//==================================================================================================
//							Beckhoff Automation Poland
//									14.03.2023
//
// Code owner: TG
//
// Function block for processing digital outputs. 
// Includes filters, simulating, various operational modes selection and edges detection.
//
// Used libraries: 
//	Tc2_standard						|| 3.3.3.0
//
// Used FBs:
//
// Used DUTs:
//
//  v1.0	|| TC v 3.1.4024.40		|| First edition
//==================================================================================================
FUNCTION_BLOCK FB_DigitalOutput
VAR
	Out 					AT %Q* 				: BOOL;
	bManualIn									: BOOL;		// HMI
	
	{attribute 'hide'}
	bManualMode_Internal						: BOOL;		// Internal flag - active when manual mode selected
	_bIn										: BOOL;
	{attribute 'hide'}
	_bOut										: BOOL; 
	{attribute 'hide'}
	_tTimeDelay									: TIME;
	{attribute 'hide'}
	_tTimeOn									: TIME;
	{attribute 'hide'}
	_tTimeOff									: TIME;
	{attribute 'hide'}
	_nMode										: DINT;															
END_VAR

CASE nMode OF							//case regarding mode selection 

	0:	// false
		Off();
	
	1:	// true
		On();

	2:	// auto normal
		Auto();
		
	9:	// manual
		Manual();
	
	10:	// clock
		Clock();

	11: // min OFF, min ON	
		MinOnOff();	
	
	20: // single TP
		SingleTP();
	
	21: // single TON
		SingleTON();	
							
	30: // mutli TP
		MultiTP();

	31:	// mutli TON
		MultiTON();
		
ELSE		
	Off();
	
		
END_CASE;

METHOD Auto 									: BOOL							//output actual value 
VAR_INPUT
END_VAR
bOut											:= bIn;

bManualMode_Internal							:= FALSE;
END_METHOD

PROPERTY bIn 									: BOOL								//value before processing
GET
bIn												:=_bIn;
END_GET
SET
_bIn											:= bIn;
END_SET
END_PROPERTY

PROPERTY bOut 									: BOOL							//processed output value
GET
bOut											:= _bOut;
END_GET
SET
_bOut											:= bOut;
Out												:= bOut;
END_SET
END_PROPERTY

METHOD Clock 									: BOOL							//use output for specifed time with pause between
VAR_INST
	{attribute 'hide'}
	tonTimer									: TON;
END_VAR
tonTimer(IN := NOT tonTimer.Q,
		PT										:= tTimeOn + tTimeOff);
bOut											:= tonTimer.ET <  tTimeOn;
		
bManualMode_Internal							:= FALSE;
END_METHOD

METHOD Manual 									: BOOL							//Control output value manually
IF bManualMode_Internal THEN
	bOut										:= bManualIn;
ELSE
	bManualIn									:= bOut;
END_IF

bManualMode_Internal							:= TRUE;
END_METHOD

METHOD ManualEx 								: BOOL							//Control output value manually
VAR_INPUT
	bIn											: BOOL;
END_VAR
bOut											:= bIn;

bManualMode_Internal							:= FALSE;
END_METHOD

METHOD MinOnOff 								: BOOL						//output with specific active and disabled time
VAR_INST
	TimeMinOn									: TON;
	TimeMinOff									: TON;	
END_VAR
TimeMinOff(IN := NOT bOut, PT := tTimeOff);			
                        						
TimeMinOn(IN := bOut, PT := tTimeOn);	
		
IF TimeMinOn.Q THEN
	bOut										:= bIn;
END_IF;			
		
IF TimeMinOff.Q THEN
	bOut										:= bIn;
END_IF;

bManualMode_Internal							:= FALSE;
END_METHOD

METHOD MultiTON 								: BOOL						//activation delay dependent from value
VAR_INST
	Timer										: TON;
END_VAR
Timer(IN := bIn, PT := tTimeDelay);

bOut											:= Timer.Q;

bManualMode_Internal							:= FALSE;
END_METHOD

METHOD MultiTP 									: BOOL							//pulse dependent from value
VAR_INST
	Timer										: TP;
END_VAR
Timer(IN := bIn, PT := tTimeOn);
		
bOut											:= Timer.Q;

bManualMode_Internal							:= FALSE;
END_METHOD

PROPERTY nMode 									: DINT							//mode selection value: 0- false 1-true 2 - auto_normal, 10- clock, 20 - single tp, 21 - single ton, 9 - manual, 30 - multi tp, 31 - multi ton, 11 - min ON, min OFF
GET
nMode											:= _nMode;
END_GET
SET
_nMode											:= nMode;
END_SET
END_PROPERTY

METHOD Off 										: BOOL								//set value FALSE
bOut											:= FALSE;

bManualMode_Internal							:= FALSE;
END_METHOD

METHOD On 										: BOOL								//set value TRUE
bOut											:= TRUE;

bManualMode_Internal							:= FALSE;
END_METHOD

METHOD SingleTON 								: BOOL						//activation delay 
VAR_INST
	Timer										: TON;
END_VAR
Timer(IN := TRUE, PT := tTimeDelay);

bOut											:= Timer.Q;

bManualMode_Internal							:= FALSE;
END_METHOD

METHOD SingleTP 								: BOOL						//single pulse
VAR_INST
	Timer										: TP;
END_VAR
Timer(IN := TRUE, PT := tTimeOn);

bOut											:= Timer.Q;

bManualMode_Internal							:= FALSE;
END_METHOD

PROPERTY tTimeDelay  								: TIME						//delay time in [ms], for Single/MultiTON mode
GET
tTimeDelay										:= _tTimeDelay;
END_GET
SET
_tTimeDelay										:= tTimeDelay;
END_SET
END_PROPERTY

PROPERTY tTimeOff 								: TIME						//minimum output on time [ms], for minOnOff mode
GET
tTimeOff										:= _tTimeOff;
END_GET
SET
_tTimeOff										:= tTimeOff;
END_SET
END_PROPERTY

PROPERTY tTimeOn 								: TIME						//minimum output off time [ms], for minOnOff mode
GET
tTimeOn											:=_tTimeOn;
END_GET
SET
_tTimeOn										:= tTimeOn;
END_SET
END_PROPERTY

END_FUNCTION_BLOCK

(* stored: Version 1.1.0.1, FileIdentifier 9c9296da76f6555697687ec98103123ce9290b24, FileSignature 4b7ff2dcf8c12612268e668eaf2997718c55023cd67da2f5992bdf710eefc9968962d0b293f44ff252512e4510ae557b74a6a527a16271f1788755e7e6d9445defe0fe348b14a65da049c3d86c0c9e8fdd809d3d46764a5bcdca4ca8c0c737abe1dca42b05d38a2eedf13d4ff265bcc4314e1f238197d24dcd4ab5bd84eb4ef6208a6f210ed1960d85d639d221da18380a7ed45771d073b4f8f16abf18f4a0101355f8787fddc439370796d36f83c19f69321c38f61acdb8ad15c808a511caa439041c93119310479aa3316171e14b610b326d88d603c3c53c91d3b49ea8358598d3b6d06331ac0704becd62f57d1ee26a41c64ff01206e21afefac73dbd0c3d
   POU FB_DigitalOutput: Id {b9e9f56b-5870-4da1-94e5-b2a4388e6247}, SpecialFunc None
   Folder Methods: Id {b5b59953-258d-4858-9d8c-ded201c1d6be}
   Folder Properties: Id {efc33531-5806-48f9-8d32-ec1e9a918ec5}
   Method Auto: Id {160ef08d-1b1b-47be-ba82-329dc9f601ad}
   Property bIn: Id {2bee2410-9535-4e3a-b7ae-806cc45d26d3}
   Get Get: Id {369e7bce-9d6f-485e-a22d-3e3080567aae}
   Set Set: Id {986d5f7b-a3f9-43b2-9906-2401471bc586}
   Property bOut: Id {a288c155-be43-44cf-b5c3-5eb498f187ba}
   Get Get: Id {25156acb-f4c8-492d-8acf-3e9d085f468c}
   Set Set: Id {fff5618d-e23c-4375-b0e7-62568e20ec8c}
   Method Clock: Id {69075f1c-9b57-4993-a762-5981a09070c3}
   Method Manual: Id {65e61266-7bcd-4120-85c8-f2b1105e0e4b}
   Method ManualEx: Id {746ecf17-5a39-4746-adb4-1e5aaf6be40d}
   Method MinOnOff: Id {b3caaa05-6ef4-4de3-9475-35763e6acaca}
   Method MultiTON: Id {cc88a96c-69ed-48a9-9728-ddfc6a7abe6b}
   Method MultiTP: Id {36ab7aad-cbc7-419a-9f0c-9c5301704b53}
   Property nMode: Id {724ef173-819e-4fa1-9b71-08b994bff2d7}
   Get Get: Id {0a2f5de2-7444-4a32-aaca-d4fad073e1d2}
   Set Set: Id {4b3056da-3dc2-46c4-a769-48c26f666f49}
   Method Off: Id {07366ab7-5d08-40f0-aa73-80842a29b190}
   Method On: Id {15dc5094-ea12-43e0-8421-88745f8eec4f}
   Method SingleTON: Id {fc60e54b-09f2-4088-8a6a-d39e5e545ee6}
   Method SingleTP: Id {c938c52e-1855-4129-8417-a709116ecb22}
   Property tTimeDelay: Id {2f3dcb9a-b10f-46bf-948d-cecc8705f27f}
   Get Get: Id {a8e48e37-318f-4723-842f-5b667fb87b93}
   Set Set: Id {31b5c6fd-c05a-43ef-bead-7d5de28e1867}
   Property tTimeOff: Id {8b3761a2-1bf1-486b-a4af-3320378b9a1f}
   Get Get: Id {f552e05c-dbe0-467a-a5b8-2fe76fc5154a}
   Set Set: Id {2141f521-0fa1-4712-aab3-f4bd11911aaa}
   Property tTimeOn: Id {59985f36-3abd-423a-9121-57dfab1fac97}
   Get Get: Id {fa200f2d-b633-4cc5-9da6-72f42c083e25}
   Set Set: Id {a4549a01-0e47-44d9-8d31-ab34193c9c2f} *)
